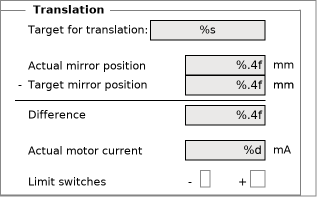
VISUALIZATION VISU_M3TranslationDetails  // 317x197
VAR_IN_OUT
	ref : M3Translation;
END_VAR
    Label (25,56 125x20), "Actual mirror position"
    Label (25,75 125x20), "Target mirror position"
    Label (30,0 150x20), "Translation"
    Label (270,55 35x20), "mm"
    Label (270,75 35x20), "mm"
    Label (25,105 150x20), "Difference"
    Label (270,75 45x20), "mm"
    Line (15,100) (265,100)
    Rectangle (185,55 80x20), "%.4f", text variable: ref.actualPosition.millimeters.value
    Rectangle (185,75 80x20), "%.4f", text variable: ref.target.position.millimeters.value
    Rectangle (185,105 80x20), "%.4f", text variable: ref.actualPositionError.millimeters.value
    Label (15,75 10x20), "-"
    Label (25,141 190x20), "Actual motor current"
    Label (270,140 35x20), "mA"
    Rectangle (185,140 80x20), "%d", text variable: ref.parts.motorDrive.averageCurrent.milliAmps.value
    Rectangle (150,20 115x20), "%s", text variable: ref.target.actualStatus
    Label (25,20 125x20), "Target for translation:"
    Label (25,172 130x20), "Limit switches"
    Label (185,172 15x20), "-"
    Frame (200,170 10x17)
        shows VISU_State_gray_red(state := ref.negativeLimitSwitchActive)
    Label (235,172 15x20), "+"
    Frame (250,170 15x17)
        shows VISU_State_gray_red(state := ref.positiveLimitSwitchActive)
    Polyline (110,10) (300,10) (300,195) (0,195) (0,10) (25,10)
END_VISUALIZATION

(* stored: Version 1.1.0.1, ProductVersion 3.1.4019.2
   Visu VISU_M3TranslationDetails: Id {e21eaa32-abf9-4b86-b441-ff37f4659ce7} *)
